//KalmanObserver:
//Implements a Kalman observer which fuses the camera measurement (measurement noise) and encoder data (process noise) to observe the position of the robot.
// Adaptive because the covariance matrix Q is a weighted mean of the covariance measurements matrices respetively to the current velocities

FUNCTION_BLOCK AdaptiveKalmanObserverST
VAR_INPUT
	xCameraPose:	RobotPoseSimple;
	xVxRobot: 		LREAL;	//measured velocities
	xVyRobot: 		LREAL;
	xOmegaRobot: 	LREAL;
	theta:			LREAL; //theta for I/O Lineraztion only explicitly Input for FF-Linearization;
END_VAR

VAR_OUTPUT
	yObserverdPose: 	RobotPoseSimple;
END_VAR

VAR
	newCamDataArrived: BOOL;
	camDataOld, observerError, observedPosition, vWorld: RobotPoseSimple;
	pulseGenerator: TP;
	
	delayedCycles		AT%Q* 	: INT	:= ControlParameters.kObsDelayedCycles;	//Camdelay 160ms / Cycletyme 2ms
	delayedPosition: ARRAY [0..140] OF RobotPoseSimple;
											
	P, H, TEMP : ARRAY [0..2,0..2] OF LREAL;

	Q : ARRAY [0..2,0..2] OF LREAL 		:=ControlParameters.Q;
											  
	RMat : ARRAY [0..2, 0..2] OF LREAL 	:= ControlParameters.RMat;
											
	C : ARRAY [0..2,0..2] OF LREAL 		:=[1, 0, 0,
    									   0, 1, 0,
   										   0, 0, 1];

	observedPositionAP: RobotPoseSimple;
	PAP: ARRAY [0..2, 0..2] OF LREAL;
	scaledCovMatX: INT;
	multiplierX: LREAL;
	scaledCovMatT: ARRAY [0..2, 0..2] OF LREAL;
	multiplierT: LREAL;
	QT1: ARRAY [0..2, 0..2] OF LREAL;
END_VAR

//transform roboter velocities into world velocities and pass them to Simulink
Robot2World( 
	vx_robot 	:= xVxRobot,
	vy_robot 	:= xVyRobot,
	omega_robot := xOmegaRobot,
	theta		:= yObserverdPose.theta,
	vx_world 	=> vWorld.x,
	vy_world  	=> vWorld.y,
	omega_world => vWorld.theta);
	
CheckForNewCameraData();	//Schreibt direkt in Variable  "newCamDataArrived"

delayPosition();

Q := calculateQMatrix();

// Step 1 Prediction
observedPositionAP := AddRPS(observedPosition, ScaleRPS(c := Var_HAWIno.CONTROLLER_CYCLE_TIME, vWorld));
PAP := AddMat3(P, Q);

//if valid cam data arrived
IF newCamDataArrived THEN
	//Step 2 Optimize H
	TEMP := AddMat3(PAP,RMat);
	TEMP := MatInv3(TEMP);
	H := MatTimesMat(PAP, TEMP);
	
	//step 3 Correction
	//calculate observer error
	observerError := SubtractRPS(xCameraPose,delayedPosition[delayedCycles]);
	//correct observed position
	observedPosition := AddRPS(observedPositionAP, MatTimesRPS(H, observerError));
	//correct obersvation covariance
	P := SubstractMat3(PAP, MatTimesMat(H, PAP));
ELSE 
	observedPosition := observedPositionAP;
	P := PAP;
END_IF

//set Outputs
yObserverdPose 	:= observedPosition;
camDataOld 		:= xCameraPose;

METHOD calculateQMatrix : ARRAY [0..2,0..2] OF LREAL
VAR_INPUT
	
END_VAR

VAR
	scaledCovMatX, scaledCovMatY, scaledCovMatT, tempMat : ARRAY[0..2,0..2] OF LREAL;
	multiplierX, multiplierY, multiplierT : LREAL;
	
	vXRef,vYRef : LREAL := 300;
	vTRef : LREAL := 1;
	
	QT1 : ARRAY[0..2,0..2] OF LREAL :=[0.7645,	-0.2488,	0.0015,
									  -0.2488,	1.0596,		-0.0026,
									  0.0015,	-0.0026,	0.0007];
									  
	QY300 : ARRAY[0..2,0..2] OF LREAL :=[1.5214,	0.3889,		0.0002,
										 0.3889,	26.0708,	-0.0210,
										 0.0002,	-0.0210,	0.0003];
										 
	QX300 : ARRAY[0..2,0..2] OF LREAL :=[9.3047,	1.1844,		-0.0125,
										 1.1844,	1.0394,		0.0001,
										 -0.0125,	0.0001,		0.0001];
END_VAR
// Calcualte Factor current vRef to vMeasurement from evaluating Covariances
multiplierX := xVxRobot / vXRef;
multiplierY := xVyRobot / vYRef;
multiplierT := xOmegaRobot / vTRef;

//Multiply respective Matrix with multiplier
scaledCovMatX := MultiplyMatrix3(multiplier:=multiplierX, matrix:= QX300);
scaledCovMatY := MultiplyMatrix3(multiplier:=multiplierY, matrix:= QY300);
scaledCovMatT := MultiplyMatrix3(multiplier:=multiplierT, matrix:= QT1);

//Calculate mean
tempMat := AddMat3(mat1:=scaledCovMatX, mat2:=scaledCovMatY);
tempMat := AddMat3(mat1:=tempMat, mat2:= scaledCovMatT);
Q := MultiplyMatrix3(matrix:=tempMat, multiplier:=0.3333);	//Set new Q directly in Kalman FB
END_METHOD

METHOD checkForNewCameraData : BOOL
VAR_INPUT
END_VAR
newCamDataArrived := (camDataOld.x <> xCameraPose.x OR camDataOld.y <> xCameraPose.y OR camDataOld.theta <> xCameraPose.theta) //cahnge in one of the positions
					 AND xCameraPose.x <> 0 AND xCameraPose.y <> 0;		//valid data
END_METHOD

METHOD PRIVATE delayPosition : BOOL
VAR_INPUT
END_VAR
VAR
	i: INT := 0;
END_VAR
FOR i := 0 TO delayedCycles-1 DO
	delayedPosition[i+1] := delayedPosition[i];
END_FOR
delayedPosition[0] := observedPosition;
END_METHOD

METHOD reset : BOOL
VAR_INPUT
END_VAR
VAR
	
END_VAR
reset := FALSE;
IF newCamDataArrived THEN
	observedPosition := xCameraPose;
	reset := TRUE;
END_IF
END_METHOD

END_FUNCTION_BLOCK

(* stored: Version 1.1.0.1, ProductVersion 3.1.4024.11
   POU AdaptiveKalmanObserverST: Id {1186a501-be3f-4ebc-9c38-7ef7659d2773}, SpecialFunc None
   Method calculateQMatrix: Id {27a638c4-8125-4fe1-9f4c-e71da7ebacf0}
   Method checkForNewCameraData: Id {1b408c7c-3602-4583-a07d-63fd82822918}
   Method delayPosition: Id {cc016d51-b2c3-42d5-96b7-225e88728129}
   Method reset: Id {ba4df63c-4587-4dcd-ac73-d64764d2f997} *)
